GLOBALCONSTANTS DefaultPool_Dreieck (* Global constants *)
  PACKAGE Uebungen::const::UT::Dreieck;
  VAR_GLOBAL CONSTANT
    ISO_DESIGNATOR_WIDTH : UINT := 80;
    ISO_DESIGNATOR_HEIGHT : UINT := 80;
    ISO_MASK_SIZE : UINT := 480;
    ISO_VERSION_LABEL : STRING;
    MASK_WIDTH : UINT := 480;
    MASK_HEIGHT : UINT := 480;
    WorkingSet : UINT := 0;
    DataMask_M1 : UINT := 1000;
    Container_Sollwertmarker : UINT := 3000;
    InputNumber_Sollwert : UINT := 9000;
    InputNumber_Istwert : UINT := 9001;
    InputNumber_Messwert : UINT := 9002;
    OutputString_WorkingSet_0 : UINT := 11000;
    OutputString_UP : UINT := 11001;
    OutputString_DOWN : UINT := 11002;
    Polygon_Bargraph_Mittelmarker : UINT := 16000;
    LinearBargraph : UINT := 18000;
    Bargraph_Split_links : UINT := 18001;
    Bargraph_Split_rechts : UINT := 18002;
    NumberVariable_Sollwert : UINT := 21000;
    NumberVariable_Istwert : UINT := 21001;
    NumberVariable_Messwert : UINT := 21002;
    FontAttributes_6x8 : UINT := 23000;
    FontAttributes_Werte : UINT := 23001;
    LineStyle_Bargraph_Mittelmarker_Gruen : UINT := 24000;
    FillStyle_Bargraph_Mittelmarker_Gruen : UINT := 25000;
  END_VAR
END_GLOBALCONSTANTS
